# EPICS SNL sequencer program: sources/expClearanceSNC.stt
program expClearanceSNC

%{
#include "vcs_var_mes.h" // define this here so C functions are seen

#define	VCOK       	0
#define TOUT		5
#define FAIL		-1
#define	EXPPNK 		19
#define RA12ON 		147
#define	DA12ON		68
#define	DA12S1OFF	75
#define	DA12S2OFF	76
#define	G9ON		151
#define	G10ON		152
#define	G9OFF		153
#define	G10OFF		154
#define B26ON		69
#define B27OFF		72
#define B28aOFF		73
#define B28bOFF		74
#define B27ON		78
#define B28aON		79
#define B28bON		80
#define B29OFF		77
}%
/* Declare seq variables*/
short EXP_INIT;
short EXP_VC;
short EXP_W26_STS;
short EXP_W28b_STS;
short EXP_W28a_STS;
short EXP_W27_STS;
short EXP_W29_STS;
short EXP_G10_STS;

short EXP_FAIL_COND;
short EXP_OLD_FAIL_COND;

string EXP_CLR_STATS;
string EXP_INTLCK_STATS;

short expUpdate= FALSE;
/* Associate SNL variables with epics output pv's*/
assign	EXP_CLR_STATS		to	"{SYS}:EXP-CLR-STATS";
assign	EXP_INTLCK_STATS	to	"{SYS}:EXP-INTLCK-STATS";
/* Associate SNL variables with epics input pv's*/
assign 	EXP_VC 				to 	"{SYS}:EXP-VC";
assign 	EXP_INIT 			to 	"{SYS}:EXP-INIT";

assign 	EXP_W26_STS 		to 	"{SYS}:EXP-W26-STS";
assign 	EXP_W28b_STS 		to  "{SYS}:EXP-W28b-STS";
assign 	EXP_W28a_STS 		to 	"{SYS}:EXP-W28a-STS";
assign 	EXP_W27_STS 		to  "{SYS}:EXP-W27-STS";
assign 	EXP_W29_STS 		to 	"{SYS}:EXP-W29-STS";
assign 	EXP_G10_STS 		to 	"{SYS}:EXP-G10-STS";
assign	EXP_FAIL_COND		to	"{SYS}:EXP-FAIL-COND";

monitor	EXP_VC;
monitor EXP_W26_STS;
monitor EXP_W28b_STS;
monitor EXP_W28a_STS;
monitor EXP_W27_STS;
monitor EXP_W29_STS;
monitor EXP_G10_STS;
monitor	EXP_FAIL_COND;

ss EXP_clearance_status {
    state init {
		when (delay(2)) {
			initVault();
			printf("\n%sEXPERIMENTAL BEAM LINE INITIALISATION COMPLETED%s\n",OK,DEF);
		} state watchman_26_pressed
    }
///////////////////////////////////////////////////////////////
	/*VAULT CLEARED STATE*/
    state vault_cleared {
		option -e;
		entry {
			printf("%sEXPERIMENTAL BEAM LINE IN CLEARED STATE%s\n",CLR,DEF);
		}
		when (EXP_VC != VCOK) {

		} state vc_faillures
	}
//////////////////////////////////////////////////////////
	state recover_faillure {

		when (EXP_FAIL_COND != EXP_OLD_FAIL_COND) {

		} state  clearance_faillures

		when (EXP_W26_STS != FAIL) {
			if(!expUpdate) {
				printf("%sEXP RECOVERING FROM FAILLURE - ENTERING W26 STATE%s\n",OK,DEF);
				expUpdate= TRUE;
			}
		} state  watchman_26_pressed

	}
//////////////////////////////////////////////////////////
	state watchman_26_pressed {
		/*option -e;
		entry {
		printf("%sEXP LAST FAILLURE: %d%s\n",OK,EXP_W26_STS,DEF);

		}*/
		when (EXP_W26_STS == FAIL) {
			EXP_OLD_FAIL_COND = EXP_FAIL_COND;
		} state  clearance_faillures

		when (EXP_W26_STS == B26ON) {
			EXP_clear_underway();
			EXP_update_report(B26ON);
		} state watchman_26_released
	}
//////////////////////////////////////////////////////////
	state watchman_26_released {

		when (EXP_W26_STS == FAIL) {

		} state  clearance_faillures

		when (EXP_W26_STS != B26ON) {
			EXP_update_report(G10OFF);
		} state gate_g10_closed
	}
//////////////////////////////////////////////////////////
	state gate_g10_closed {

		when (EXP_W26_STS == FAIL) {

		} state  clearance_faillures

		when (!EXP_G10_STS) {
			EXP_update_report(B28bOFF);
		} state watchman_28b_pressed
	}
//////////////////////////////////////////////////////////
	state watchman_28b_pressed {

		when (EXP_W26_STS == FAIL) {

		} state   clearance_faillures

		when (EXP_W28b_STS == B28bON) {
			EXP_update_report(B28bON);
		} state watchman_28b_released
	}
//////////////////////////////////////////////////////////
	state watchman_28b_released {

		when (EXP_W26_STS == FAIL) {

		} state  clearance_faillures

		when (EXP_W28b_STS != B28bON) {
			EXP_update_report(B28aOFF);
		} state watchman_28a_pressed
	}
///////////////////////////////////////////////////////////
	state watchman_28a_pressed {

		when (EXP_W26_STS == FAIL) {

		} state  clearance_faillures

		when (EXP_W28b_STS == B28aON) {
			EXP_update_report(B28aON);
		} state watchman_28a_released
	}
//////////////////////////////////////////////////////////
	state watchman_28a_released {

		when (EXP_W26_STS == FAIL) {

		} state  clearance_faillures

		when (EXP_W28b_STS != B28aON) {
			EXP_update_report(B27OFF);
		} state watchman_27_pressed
	}
///////////////////////////////////////////////////////////
	state watchman_27_pressed {

		when (EXP_W26_STS == FAIL) {

		} state  clearance_faillures

		when (EXP_W27_STS == B27ON) {
			EXP_update_report(B27ON);
		} state watchman_27_released
	}
//////////////////////////////////////////////////////////
	state watchman_27_released {

		when (EXP_W26_STS == FAIL) {

		} state  clearance_faillures

		when (EXP_W27_STS != B27ON) {

		} state door_a12_closed
	}
//////////////////////////////////////////////////////////
	state door_a12_closed {

		when (EXP_W26_STS == FAIL) {

		} state  clearance_faillures

		when (EXP_W29_STS == DA12S1OFF) {
			EXP_update_report(DA12S1OFF);
		} state door_a12_closed

		when (EXP_W29_STS == DA12S2OFF) {
			EXP_update_report(DA12S2OFF);
		} state door_a12_closed

		when () {
			EXP_update_report(B29OFF);
		} state watchman_29_pressed
	}
///////////////////////////////////////////////////////////
	state watchman_29_pressed {

		when (EXP_W26_STS == FAIL) {

		} state  clearance_faillures

		when (!EXP_W29_STS) {

			EXP_status();
		} state vault_cleared
	}
//////////////////////////////////////////////////////////////////
	state clearance_faillures { 			/* FAIL CONDITIONS*/

		option -e;
		option -x;
		entry {
			printf("EXP CLEARANCE FAILURE CONDITION: ");
			expUpdate = FALSE;
			EXP_OLD_FAIL_COND = EXP_FAIL_COND;
		}

		when (EXP_FAIL_COND == RA12ON) {
			EXP_update_failed(RA12ON);
			printf("%sROOF A12 IS OPEN%s\n",ERROR,DEF);
		} state recover_faillure

		when (EXP_FAIL_COND == TOUT) {
			EXP_update_failed(TOUT);
			printf("%sTIME OUT ERROR: RELEASE ALL WATCHMEN%s\n",ERROR,DEF);
		} state recover_faillure

		when () {
		} state gate_faillures

		exit {
		    EXP_OLD_FAIL_COND = EXP_FAIL_COND;
		}

	}
//////////////////////////////////////////////////////////////////
	state gate_faillures { 			/* DOOR A1A FAIL CONDITIONS*/

		option -x;

		when (EXP_FAIL_COND == G9ON) {
			EXP_update_failed(G9ON);
			printf("%sGATE G9 WAS OPENED%s\n",ERROR,DEF);
		} state recover_faillure

		when (EXP_FAIL_COND == G10ON) {
			EXP_update_failed(G10ON);
			printf("%sGATE G10 WAS OPENED%s\n",ERROR,DEF);
		} state recover_faillure

		when () { // THIS MAY NOT BE NECCESSARY
		} state recover_faillure

		exit {
		    EXP_OLD_FAIL_COND = EXP_FAIL_COND;
		}
	}
////////////////////////////////////////////////////////////////////////////
	state vc_faillures { 			/* FAIL CONDITIONS*/

		option -e;
		option -x;
		entry {
			printf("EXP LOW CLEAR FAILURE CONDITION: ");
			expUpdate = FALSE;
		}

		when (EXP_VC == RA12ON) {
			EXP_update_failed(RA12ON);
			printf("%sROOF A12 IS OPEN%s\n",ERROR,DEF);
		} state recover_faillure

		when (EXP_VC == G9ON) {
			EXP_update_failed(G9ON);
			printf("%sGATE G9 WAS OPENED%s\n",ERROR,DEF);
		} state recover_faillure

		when (EXP_VC == G10ON) {
			EXP_update_failed(G10ON);
			printf("%sGATE G10 WAS OPENED%s\n",ERROR,DEF);
		} state recover_faillure

		when (EXP_VC == DA12ON) {
			EXP_update_failed(DA12ON);
			printf("%sDOOR A12 WAS OPENED%s\n",ERROR,DEF);
		} state recover_faillure

		when (EXP_VC == EXPPNK) {
			EXP_update_failed(EXPPNK);
			printf("%sA PANIC BUTTON WAS  PRESSED%s\n",ERROR,DEF);
		} state recover_faillure

		exit {
		    EXP_OLD_FAIL_COND = EXP_FAIL_COND;
		}
	}
}

void initVault(){
	EXP_INIT = TRUE;
	not_cleared(EXP_CLR_STATS);
	report_error(EXP_INTLCK_STATS, 54);
	pvPut(EXP_INIT, SYNC);
	pvPut(EXP_CLR_STATS, SYNC);
	pvPut(EXP_INTLCK_STATS, SYNC);
	EXP_OLD_FAIL_COND = EXP_FAIL_COND;
}

void resetStatus()
{
	not_cleared(EXP_CLR_STATS);
	report_error(EXP_INTLCK_STATS, 54);
	pvPut(EXP_CLR_STATS, SYNC);
	pvPut(EXP_INTLCK_STATS, SYNC);
}
////////////////////////////////////////////////////////////////////////
void EXP_update_failed(short report)
{
	clear_failed(EXP_CLR_STATS);
	pvPut(EXP_CLR_STATS, SYNC);
	report_error(EXP_INTLCK_STATS, report);
	pvPut(EXP_INTLCK_STATS, SYNC);
}
/////////////////////////////////////////////////////////////////////////
void EXP_update_report(short intlck) {
	report_error(EXP_INTLCK_STATS, intlck);
	pvPut(EXP_INTLCK_STATS, SYNC);
}
////////////////////////////////////////////////////////////////////////
void EXP_status()
{
	cleared(EXP_CLR_STATS);
	pvPut(EXP_CLR_STATS, SYNC);
	report_error(EXP_INTLCK_STATS, 54);
	pvPut(EXP_INTLCK_STATS, SYNC);
}
///////////////////////////////////////////////////////////
void EXP_clear_underway()
{
	clear_underway(EXP_CLR_STATS);
	pvPut(EXP_CLR_STATS, SYNC);
}
/**********************************************************/
